FUNCTION HEXSTR_TO_REAL_LHeaterPV : REAL
VAR_INPUT
	hStrTemperaturePV : STRING;
END_VAR
VAR
	hData			:UDINT;
	aData	: ARRAY[0..1]OF BYTE;
	bSwap	: BYTE;
	ptStrTemperature : POINTER TO INT;
	nTemperaturePV : INT;
END_VAR

// Convert to Data Array from HexString
hData := HEXSTR_TO_DATA(hStrTemperaturePV, ADR(aData), SIZEOF(aData));

//Swap Data
bSwap := aData[0];
aData[0] := aData[1];
aData[1] := bSwap;

ptStrTemperature := ADR(aData);
nTemperaturePV := ptStrTemperature^;
HEXSTR_TO_REAL_LHeaterPV := INT_TO_REAL(nTemperaturePV);

END_FUNCTION

(* stored: Version 1.1.0.1, ProductVersion 3.1.4024.12
   POU HEXSTR_TO_REAL_LHeaterPV: Id {07cfba14-5fdf-48c5-9c53-d8abb8f4ad05}, SpecialFunc None *)
